{attribute 'c++_compatible'} 
FUNCTION_BLOCK ARCommunicationMQTTExtention_t EXTENDS FB_IotMqttClient
VAR_INPUT
END_VAR
VAR_OUTPUT
END_VAR

VAR
	_newMessageAvalable : BOOL := FALSE;	

	(* received message *)
	{attribute 'TcEncoding':='UTF-8'}
	sTopicRcv : STRING(255);
	{attribute 'TcEncoding':='UTF-8'}
	sPayloadRcv : STRING(255);
END_VAR

METHOD getPayload : STRING(255)
{attribute 'c++_compatible'}
VAR_INPUT
END_VAR
getPayload := sPayloadRcv;
return;
END_METHOD

PROPERTY newMessageAvalable : BOOL
{attribute 'c++_compatible'}
GET
{attribute 'c++_compatible'}
VAR
END_VAR
newMessageAvalable := _newMessageAvalable;
return;
END_GET
SET
{attribute 'c++_compatible'}
VAR
END_VAR
_newMessageAvalable := newMessageAvalable;
return;
END_SET
END_PROPERTY

{attribute 'c++_compatible'}
{attribute 'pack_mode' := '4'}
{attribute 'show'}
{attribute 'minimal_input_size' := '4'}
METHOD OnMqttMessage : Tc3_IotBase.HRESULT
VAR_IN_OUT CONSTANT
	topic	: STRING;
END_VAR
VAR_INPUT
	(* pointer to payload*)
	payload	: Tc3_IotBase.PVOID;
	(* payload size in bytes*)
	length	: UDINT;
	qos	: Tc3_IotBase.TcIotMqttQos;
	repeated	: BOOL;
END_VAR

VAR
	nPayloadRcvLen : UDINT;
END_VAR
SUPER^.nMessagesRcv := SUPER^.nMessagesRcv + 1;

STRNCPY( ADR(sTopicRcv), ADR(topic), SIZEOF(sTopicRcv) );
nPayloadRcvLen := MIN(length, DINT_TO_UDINT(SIZEOF(sPayloadRcv))-1);
MEMCPY( ADR(sPayloadRcv), payload, nPayloadRcvLen );
sPayloadRcv[nPayloadRcvLen] := 0;  // ensure a null termination of received string

OnMqttMessage := S_OK;

_newMessageAvalable := TRUE;
END_METHOD

END_FUNCTION_BLOCK

(* stored: Version 1.1.0.1
   POU ARCommunicationMQTTExtention_t: Id {d1cc8469-cf02-4488-a7f1-6242361a8b0e}, SpecialFunc None
   Method getPayload: Id {9cef113e-ae9f-49da-99d6-fc09f56d6a95}
   Property newMessageAvalable: Id {6af65c4c-f13b-41dc-83c5-2406fa96aebf}
   Get Get: Id {768c67cf-5b35-4de3-a6b6-be989d2fd79a}
   Set Set: Id {525f935b-939b-4874-a503-237144bd1de8}
   Method OnMqttMessage: Id {b39d5461-55e4-4d65-9fb4-9ee8938d6d05} *)
